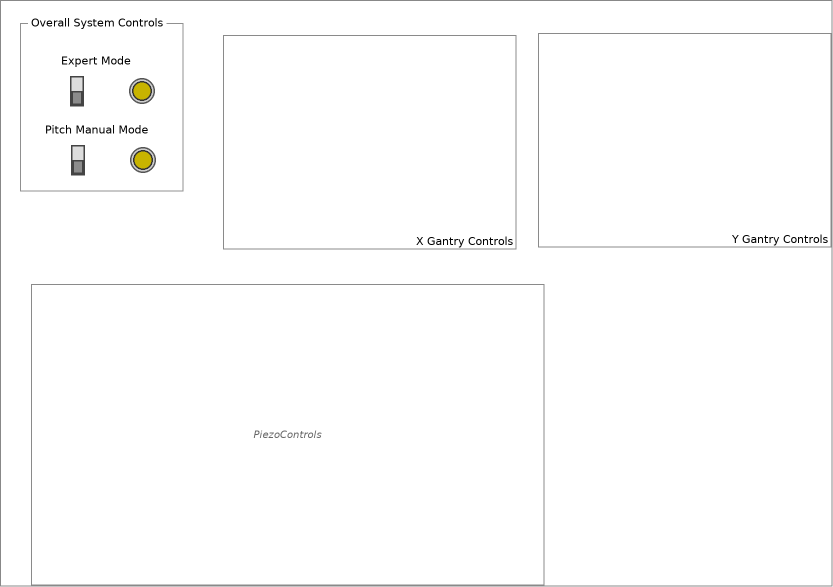
VISUALIZATION Visualization  // 833x587
    Frame (223,35 293x214), "X Gantry Controls"
        shows GantryControls(Gantry := XGantry)
    GroupBox (20,15 163x176), "Overall System Controls"
        Group (17,31 120x60)
            DipSwitch (0,30 80x30), tooltip "Puts the pitch control function block into manual mode. In manual mode the piezo and stepper movements are completely independent of one another and no coordinated actions take place. Limit switches are still respected.", variable: MAIN.ExpertMode, behaviour: TOGGLE, style: Switch-DipSwitch-Gray
            Label (3,0 112x30), "Expert Mode"
            Lamp1 (90,30 30x30), variable: MAIN.ExpertMode, style: Lamp-Lamp1-Yellow
        Group (18,100 120x60)
            DipSwitch (0,30 80x30), tooltip "Puts the pitch control function block into manual mode. In manual mode the piezo and stepper movements are completely independent of one another and no coordinated actions take place. Limit switches are still respected.", variable: MAIN.PitchManualMode, behaviour: TOGGLE, style: Switch-DipSwitch-Gray
            Label (3,0 112x30), "Pitch Manual Mode"
            Lamp1 (90,30 30x30), variable: MAIN.PitchControl.ManualMode, style: Lamp-Lamp1-Yellow
    Frame (31,284 513x301)
        shows PiezoControls(Piezo := gPitch.Piezo, ActPos := gPitch.Stepper)
    Frame (538,33 293x214), "Y Gantry Controls"
        shows GantryControls(Gantry := YGantry)
END_VISUALIZATION

(* stored: Version 1.1.0.1, ProductVersion 3.1.4020.12
   Visu Visualization: Id {2842b111-ef8a-453c-b858-3dcb33a12eaf} *)
